LIN {X 508.301, Y 346.249, Z 402.192, A -110.612, B 84.801, C -94.37, E1 0, E2 0, E3 0, E4 0}
LIN {X 507.267, Y 341.363, Z 402.642, A -110.612, B 84.801, C -94.37, E1 0, E2 0, E3 0, E4 0}
LIN {X 546.596, Y 329.892, Z 402.359, A -110.612, B 84.801, C -94.37, E1 0, E2 0, E3 0, E4 0}
LIN {X 528.42, Y 330.007, Z 402.931, A -110.612, B 84.801, C -94.37, E1 0, E2 0, E3 0, E4 0}
LIN {X 506.184, Y 336.492, Z 403.091, A -110.612, B 84.801, C -94.37, E1 0, E2 0, E3 0, E4 0}
LIN {X 505.029, Y 331.642, Z 403.541, A -110.612, B 84.801, C -94.37, E1 0, E2 0, E3 0, E4 0}
LIN {X 510.534, Y 330.036, Z 403.502, A -110.612, B 84.801, C -94.37, E1 0, E2 0, E3 0, E4 0}
PTP {X 554.276, Y 348.908, Z 474.151, A -110.612, B 84.801, C -94.37, E1 0, E2 0, E3 0, E4 0, S 'B010'}
PTP {A1 5, A2 -90, A3 100, A4 5, A5 -10, A6 -5, E1 0, E2 0, E3 0, E4 0} C_PTP
;ENDFOLD

END
